(* CODESYS project Demo_MQTT.project

Project tree, tasks and I/O mapping:
  Device : P2CDS622, AutomationDirect.com, order no. n/a, version 1.1.8.0
    application Application
      libraries: Standard, 3.5.18.0 (System); StringUtils, 3.5.20.0 (System); VisuDialogs, * (System); MQTT Client SL, 1.9.0.0 (CODESYS); Web Socket Client SL, 1.9.0.0 (CODESYS); Net Base Services, 3.5.20.0 (CODESYS); BASIC, 3.31 (OSCAT)
      task MainTask (cyclic, interval t#20ms, priority 1) calls PRG
      task VISU_TASK (cyclic, interval 100 ms, priority 31) calls VisuElems.Visu_Prg
      program PRG [CFC]
      visualisation Visualization
      text list QoSTextlist
      function TerminateString [ST]
      image pool ImagePool
      text list ModeTextList
      text list VersionTextList
    Base : P2-04B, AutomationDirect.com, order no. abc, version 1.1.8.0
      Module : P2-08SIM, AutomationDirect.com, order no. P2-08SIM, version 0.0.2
          unmapped channels: Channels
      <Empty>
      <Empty>
      <Empty>
    P2CDS622_NetConfig : P2CDS622_NetConfig, AutomationDirect.com, order no. n/a, version 1.0.0.0
        settings: ET2: IP Address = [10,201,36,189]; ET2: Subnet Mask = [255,255,255,0]
  text list GlobalTextList
  5ce3da45-db07-42e7-a21c-a00fff4ed8f6|C:\Users\a.werner\Documents\background.jpg
*)

// Device/Application/PRG
// MQTT Client with visualization
PROGRAM PRG
VAR
	mqttClient : MQTT.MQTTClient; // Function block to establish a connection to a MQTT broker
	mqttPublisher : MQTT.MQTTPublish; // Function block to publish MQTT messages
	mqttPublisher2 : MQTT.MQTTPublish; // Function block to publish MQTT messages
	mqttSubscriber : MQTT.MQTTSubscribe; // Function block to subscribe MQTT topics
	mqttSubscriber2 : MQTT.MQTTSubscribe; // Function block to subscribe MQTT topics
	sHostname : STRING(255) := 'e737de6c210d405597c25f68240b4f2b.s2.eu.hivemq.cloud'; // My HiveMQ Hostname or ip address or URL (for WebSockets: ws:// or wss://)
	uiPort : UINT := 1883; // Port of the MQTT broker
	wsPublishTopic : WSTRING(1024) := ""; // Topic to publish a message
	wsPublishTopic2 : WSTRING(1024) := ""; // Topic to publish a message
	wsSubcribeTopicFilter : WSTRING(1024) := ""; // Topic filter to subcribe a topic
	wsSubcribeTopicFilter2 : WSTRING(1024) := ""; // Topic filter to subcribe a topic
	sWillMessage : STRING(1024); // The last will message
	sPublishMessage : STRING(1024) := ''; // The messsage to publish
	sPublishMessage2 : STRING(1024) := ''; // The messsage to publish
	sSubscribeMessage : STRING(4096); // Message buffer with the retrieved message  
	sSubscribeMessage2 : STRING(4096); // Message buffer with the retrieved message  
	rsPub1Error: RS; // Helper to publisher state
	rsPub1Done: RS; // Helper to publisher state
	rsPub2Error: RS; // Helper to publisher state
	rsPub2Done: RS; // Helper to publisher state
	eCommunicationMode : MQTT.COMMUNICATION_MODE := MQTT.COMMUNICATION_MODE.TCP; // Communication mode: TCP/IP or WebSockets
	eMQTTVersion : MQTT.MQTT_VERSION := MQTT.MQTT_VERSION.V3_1_1; // The MQTT protocol version

	// Example of connect properties (V5 only)
	mQTTConnectProperties : MQTT.MQTTConnectProperties := (
		udiSessionExpiryInterval := 10,
		udiMaximumPacketSize := MQTT.MQTTParam.g_udiMaxPacketSize,
		userProperties := 
			[
				(wsKey := "key1", wsValue := "value1"),
				(wsKey := "key2", wsValue := "value2"),	
				(wsKey := "key3", wsValue := "value3")
			]
	);
	
	// Example of will properties (V5 only)
	mQTTWillProperties : MQTT.MQTTWillProperties := (
		bPayloadFormatIndicator := 1, // 1: UTF-8, 0: Binary
		wsContentType := "text/plain",
		udiMessageExpiryInterval := 60,
		udiWillDelayInterval := 60,
		userProperties := 
		[
			(wsKey := "key1", wsValue := "value1"),
		 	(wsKey := "key2", wsValue := "value2"),	
			(wsKey := "key3", wsValue := "value3")
		]);
	
	// Example of publish properties (V5 only)
	mqTTPublishProperties : MQTT.MQTTPublishProperties := (
		bPayloadFormatIndicator := 1, // 1: UTF-8, 0: Binary
		wsContentType := "text/plain",
		udiMessageExpiryInterval := 60,
		userProperties := 
		[
			(wsKey := "key1", wsValue := "value1"),
		 	(wsKey := "key2", wsValue := "value2"),	
			(wsKey := "key3", wsValue := "value3")
		]
	);
	
	// Example of subscribe properties (V5 only)
	mQTTSubscribeProperties : MQTT.MQTTSubscribeProperties := (
		udiSubscriptionIdentifier := 4343,
		userProperties := 
		[
			(wsKey := "key1", wsValue := "value1"),
		 	(wsKey := "key2", wsValue := "value2"),	
			(wsKey := "key3", wsValue := "value3")
		],
		xNoLocalOption := FALSE
	);
	
	/// If you want to use client certificates, you can configure the connection via the TLS context.
	//
	// Example (static):
	//
	// _sCommonName : STRING := 'COMMON_NAME_OF_CERTIFICATE'; // CN of the certificate (common name). 
	// _sCipherList : NBS.CIPHER_LIST := STRUCT(psList := ADR('HIGH'), udiSize := 5); // Cipher string see https://www.openssl.org/docs/man1.1.1/man1/ciphers.html
	// _ciDefaultCertInfo : NBS.CERT_INFO := (psInfo := ADR(_sCommonName), udiSize := SIZEOF(_sCommonName)); // CN of the certificate (common name)
	
	// _tlsContext : NBS.TLSContext := (	sUseCaseName := _sCommonName, // A certificate is stored in the certificate store with the use case name. You can choose any name. Here we use the common name.
	//									ePurpose := NBS.PURPOSE.CLIENT_SIDE, // For client certificates set this to NBS.PURPOSE.CLIENT_SIDE
	//									sTLSVersion := '1.2', // The TLS version
	//									sCipherList := _sCipherList, // Set the cipher list
	//									sHostname := 'HOSTNAME_OF_THE_BROKER', // The hostname of the broker
	//									udiVerificationMode := 2, // 2 => Active Peer verification
	//									ciCertInfo := _ciDefaultCertInfo, // Set the cert info
	//									itfCertVerifer := 0); // 0 => No Verifier 
	// 
	// mqttClient : MQTT.MQTTClient := (itfTLSCOntext := _tlsContext);
    //
	// You can use the method TLSContext.SetInitialValue to set the context while runtime and set the context via the input itfTLSCOntext of the client FB.
END_VAR

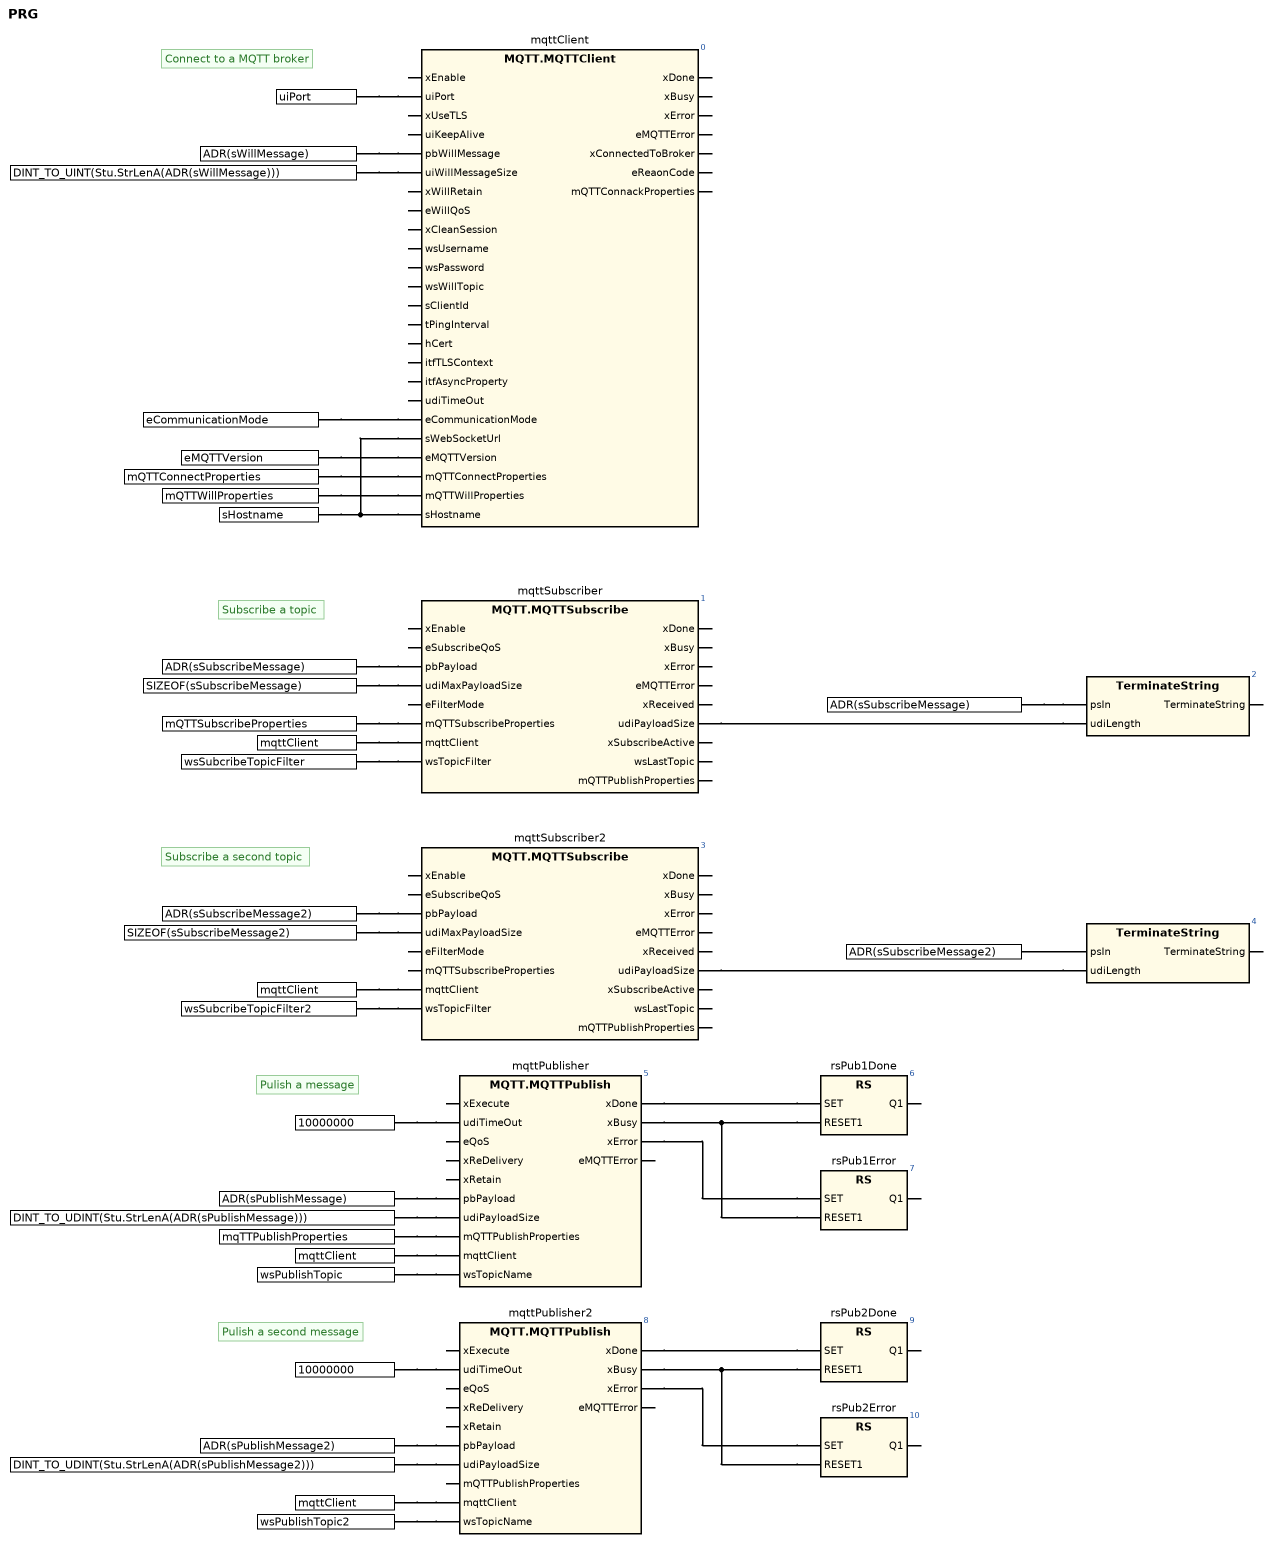
// Connect to a MQTT broker
mqttClient(
    uiPort := uiPort,
    pbWillMessage := ADR(sWillMessage),
    uiWillMessageSize := DINT_TO_UINT(Stu.StrLenA(ADR(sWillMessage))),
    eCommunicationMode := eCommunicationMode,
    sWebSocketUrl := sHostname,
    eMQTTVersion := eMQTTVersion,
    mQTTConnectProperties := mQTTConnectProperties,
    mQTTWillProperties := mQTTWillProperties,
    sHostname := sHostname); // MQTT.MQTTClient
// Subscribe a topic
mqttSubscriber(
    pbPayload := ADR(sSubscribeMessage),
    udiMaxPayloadSize := SIZEOF(sSubscribeMessage),
    mQTTSubscribeProperties := mQTTSubscribeProperties,
    mqttClient := mqttClient,
    wsTopicFilter := wsSubcribeTopicFilter); // MQTT.MQTTSubscribe
TerminateString(psIn := ADR(sSubscribeMessage), udiLength := mqttSubscriber.udiPayloadSize);
// Subscribe a second topic
mqttSubscriber2(
    pbPayload := ADR(sSubscribeMessage2),
    udiMaxPayloadSize := SIZEOF(sSubscribeMessage2),
    mqttClient := mqttClient,
    wsTopicFilter := wsSubcribeTopicFilter2); // MQTT.MQTTSubscribe
TerminateString(psIn := ADR(sSubscribeMessage2), udiLength := mqttSubscriber2.udiPayloadSize);
// Pulish a message
mqttPublisher(
    udiTimeOut := 10000000,
    pbPayload := ADR(sPublishMessage),
    udiPayloadSize := DINT_TO_UDINT(Stu.StrLenA(ADR(sPublishMessage))),
    mQTTPublishProperties := mqTTPublishProperties,
    mqttClient := mqttClient,
    wsTopicName := wsPublishTopic); // MQTT.MQTTPublish
rsPub1Done(SET := mqttPublisher.xDone, RESET1 := mqttPublisher.xBusy); // RS
rsPub1Error(SET := mqttPublisher.xError, RESET1 := mqttPublisher.xBusy); // RS
// Pulish a second message
mqttPublisher2(
    udiTimeOut := 10000000,
    pbPayload := ADR(sPublishMessage2),
    udiPayloadSize := DINT_TO_UDINT(Stu.StrLenA(ADR(sPublishMessage2))),
    mqttClient := mqttClient,
    wsTopicName := wsPublishTopic2); // MQTT.MQTTPublish
rsPub2Done(SET := mqttPublisher2.xDone, RESET1 := mqttPublisher2.xBusy); // RS
rsPub2Error(SET := mqttPublisher2.xError, RESET1 := mqttPublisher2.xBusy); // RS

END_PROGRAM

// Device/Application/TerminateString
// Terminates the STRING psIn at position udiLength
FUNCTION TerminateString : BOOL
VAR_INPUT
	psIn : POINTER TO BYTE; // Pointer to STRING
	udiLength : UDINT; // Length of psIn
END_VAR
VAR
END_VAR

psIn[udiLength] := 0;
TerminateString := TRUE;

END_FUNCTION

// Device/Application/Visualization
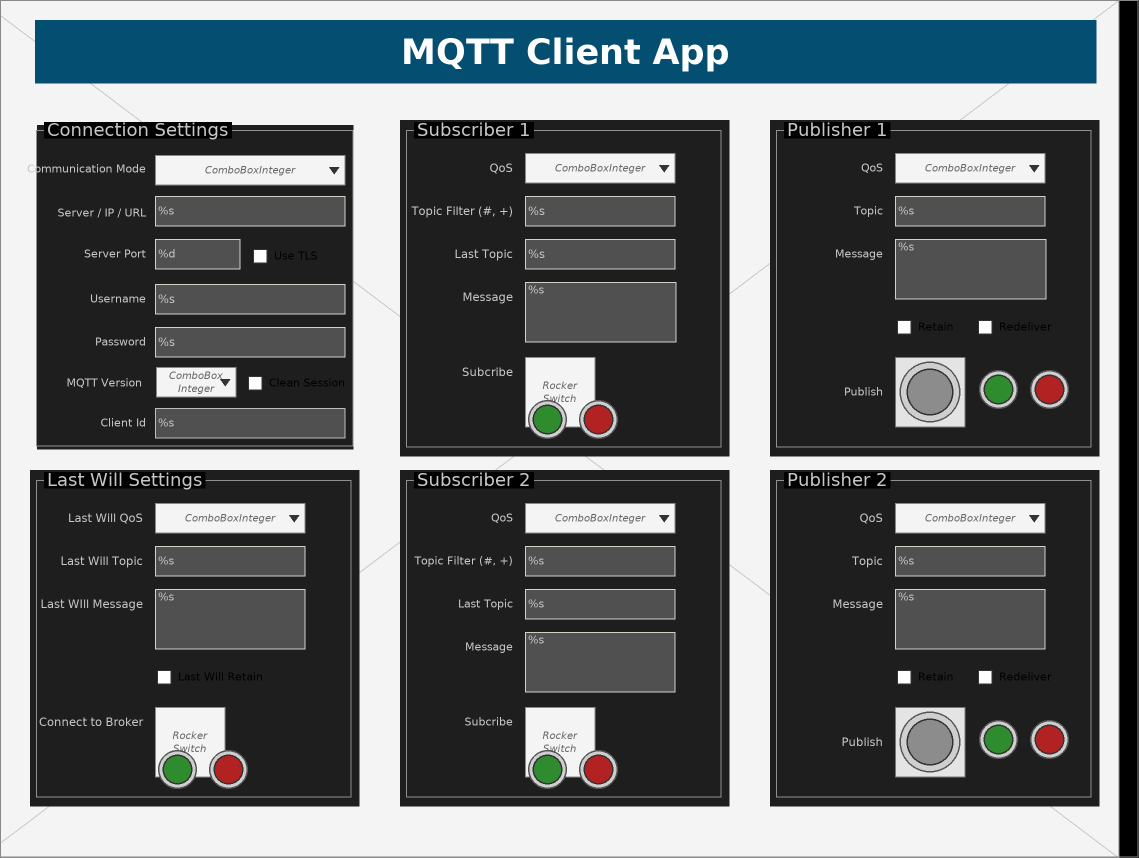
VISUALIZATION Visualization  // 1139x858
    Image (-20,0 1139x858), image: ImagePool.background
    Rectangle (37,125 316x324)
    Group (30,470 329x336)
        Rectangle (0,0 329x336)
        GroupBox (6,2 315x325), "Last Will Settings"
            ComboBoxInteger (119,31 150x30), variable: PRG.mqttClient.eWillQoS, text list: 'QoSTextlist'
        Label (16,33 100x30), "Last Will QoS"
        Textfield (125,76 150x30), "%s", text variable: PRG.mqttClient.wsWillTopic
            OnMouseClick: write the text variable via Default
        Label (16,76 100x30), "Last Will Topic"
        Textfield (125,119 150x60), "%s", text variable: PRG.sWillMessage
            OnMouseClick: write the text variable via Default
        Label (16,119 100x30), "Last WIll Message"
        Checkbox (125,192 150x30), "Last Will Retain", variable: PRG.mqttClient.xWillRetain
        Label (16,237 100x30), "Connect to Broker"
        RockerSwitch (125,237 70x70), variable: PRG.mqttClient.xEnable, behaviour: TOGGLE, style: Switch-RockerSwitch-Gray
        Lamp1 (125,277 45x45), variable: PRG.mqttClient.xConnectedToBroker, style: Lamp-Lamp1-Green
        Lamp1 (176,277 45x45), variable: PRG.mqttClient.xError, style: Lamp-Lamp1-Red
    Rectangle (770,120 329x336)
    GroupBox (776,122 315x325), "Publisher 1"
    ComboBoxInteger (895,153 150x30), variable: PRG.mqttPublisher.eQoS, text list: 'QoSTextlist'
    Label (786,153 100x30), "QoS"
    Textfield (895,196 150x30), "%s", text variable: PRG.wsPublishTopic
        OnMouseClick: write the text variable via Default
    Label (786,196 100x30), "Topic"
    Textfield (895,239 151x60), "%s", text variable: PRG.sPublishMessage
        OnMouseClick: write the text variable via Default
    Label (786,239 100x30), "Message"
    Checkbox (895,312 79x30), "Retain", variable: PRG.mqttPublisher.xRetain
    Checkbox (976,312 97x30), "Redeliver", variable: PRG.mqttPublisher.xReDelivery
    PushSwitch (895,357 70x70), variable: PRG.mqttPublisher.xExecute, input disabled if: NOT PRG.mqttClient.xConnectedToBroker, behaviour: TAP, style: Switch-PushSwitch-Gray
    Label (786,377 100x30), "Publish"
    Lamp1 (976,367 45x45), variable: PRG.rsPub1Done.Q1, style: Lamp-Lamp1-Green
    Lamp1 (1027,367 45x45), variable: PRG.rsPub1Error.Q1, style: Lamp-Lamp1-Red
    Group (770,470 329x336)
        Rectangle (0,0 329x336)
        GroupBox (6,2 315x325), "Publisher 2"
        ComboBoxInteger (125,33 150x30), variable: PRG.mqttPublisher2.eQoS, text list: 'QoSTextlist'
        Label (16,33 100x30), "QoS"
        Textfield (125,76 150x30), "%s", text variable: PRG.wsPublishTopic2
            OnMouseClick: write the text variable via Default
        Label (16,76 100x30), "Topic"
        Textfield (125,119 150x60), "%s", text variable: PRG.sPublishMessage2
            OnMouseClick: write the text variable via Default
        Label (16,119 100x30), "Message"
        Checkbox (125,192 80x30), "Retain", variable: PRG.mqttPublisher2.xRetain
        Checkbox (206,192 80x30), "Redeliver", variable: PRG.mqttPublisher2.xReDelivery
        PushSwitch (125,237 70x70), variable: PRG.mqttPublisher2.xExecute, input disabled if: NOT PRG.mqttClient.xConnectedToBroker, behaviour: TAP, style: Switch-PushSwitch-Gray
        Label (16,257 100x30), "Publish"
        Lamp1 (206,247 45x45), variable: PRG.rsPub2Done.Q1, style: Lamp-Lamp1-Green
        Lamp1 (257,247 45x45), variable: PRG.rsPub2Error.Q1, style: Lamp-Lamp1-Red
    Group (400,470 329x336)
        Rectangle (0,0 329x336)
        GroupBox (6,2 315x325), "Subscriber 2"
        ComboBoxInteger (125,33 150x30), variable: PRG.mqttSubscriber2.eSubscribeQoS, text list: 'QoSTextlist'
        Label (16,33 100x30), "QoS"
        Textfield (125,76 150x30), "%s", text variable: PRG.wsSubcribeTopicFilter2
            OnMouseClick: write the text variable via Default
        Label (16,76 100x30), "Topic Filter (#, +)"
        Textfield (125,162 150x60), "%s", text variable: PRG.sSubscribeMessage2
        Label (16,162 100x30), "Message"
        RockerSwitch (125,237 70x70), variable: PRG.mqttSubscriber2.xEnable, input disabled if: NOT PRG.mqttClient.xConnectedToBroker, behaviour: TOGGLE, style: Switch-RockerSwitch-Gray
        Label (16,237 100x30), "Subcribe"
        Lamp1 (125,277 45x45), variable: PRG.mqttSubscriber2.xSubscribeActive, style: Lamp-Lamp1-Green
        Lamp1 (176,277 45x45), variable: PRG.mqttSubscriber2.xError, style: Lamp-Lamp1-Red
        Label (16,119 100x30), "Last Topic"
        Textfield (125,119 150x30), "%s", text variable: PRG.mqttSubscriber2.wsLastTopic
    Group (400,120 329x336)
        Rectangle (0,0 329x336)
        GroupBox (6,2 315x325), "Subscriber 1"
        ComboBoxInteger (125,33 150x30), variable: PRG.mqttSubscriber.eSubscribeQoS, text list: 'QoSTextlist'
        Label (16,33 100x30), "QoS"
        Textfield (125,76 150x30), "%s", text variable: PRG.wsSubcribeTopicFilter
            OnMouseClick: write the text variable via Default
        Label (16,76 100x30), "Topic Filter (#, +)"
        Textfield (125,162 151x60), "%s", text variable: PRG.sSubscribeMessage
        Label (16,162 100x30), "Message"
        RockerSwitch (125,237 70x70), variable: PRG.mqttSubscriber.xEnable, input disabled if: NOT PRG.mqttClient.xConnectedToBroker, behaviour: TOGGLE, style: Switch-RockerSwitch-Gray
        Label (16,237 100x30), "Subcribe"
        Lamp1 (125,277 45x45), variable: PRG.mqttSubscriber.xSubscribeActive, style: Lamp-Lamp1-Green
        Lamp1 (176,277 45x45), variable: PRG.mqttSubscriber.xError, style: Lamp-Lamp1-Red
        Label (16,119 100x30), "Last Topic"
        Textfield (125,119 150x30), "%s", text variable: PRG.mqttSubscriber.wsLastTopic
    GroupBox (36,122 317x324), "Connection Settings"
        ComboBoxInteger (119,33 190x30), variable: PRG.eCommunicationMode, text list: 'ModeTextList'
        Label (-23,32 136x30), "Communication Mode"
        Textfield (119,74 190x30), "%s", text variable: PRG.sHostname
            OnMouseClick: write the text variable via Default
        Label (13,117 100x30), "Server Port", invisible if: PRG.eCommunicationMode = MQTT.COMMUNICATION_MODE.WEB_SOCKET
        Label (13,286 100x30), "Client Id"
        Textfield (119,286 190x30), "%s", text variable: PRG.mqttClient.sClientId
            OnMouseClick: write the text variable via Default
        Label (13,205 100x30), "Password"
        Textfield (119,205 190x30), "%s", text variable: PRG.mqttClient.wsPassword
            OnMouseClick: write the text variable via Default
        Label (13,162 100x30), "Username"
        Textfield (119,162 190x30), "%s", text variable: PRG.mqttClient.wsUsername
            OnMouseClick: write the text variable via Default
        Textfield (119,117 85x30), "%d", text variable: PRG.uiPort, invisible if: PRG.eCommunicationMode = MQTT.COMMUNICATION_MODE.WEB_SOCKET
            OnMouseClick: write the text variable via Default
        Label (-12,76 125x30), "Server / IP / URL"
        Checkbox (215,119 75x30), "Use TLS", variable: PRG.mqttClient.xUseTLS, invisible if: PRG.eCommunicationMode = MQTT.COMMUNICATION_MODE.WEB_SOCKET
        ComboBoxInteger (120,245 80x30), variable: PRG.eMQTTVersion, text list: 'VersionTextList'
        Label (23,246 86x30), "MQTT Version"
        Checkbox (210,246 103x30), "Clean Session", variable: PRG.mqttClient.xCleanSession
    Rectangle (35,20 1061x63), "MQTT Client App"
END_VISUALIZATION

(* text list QoSTextlist (id | default)
  0 | QoS 0
  1 | QoS 1
  2 | QoS 2
   |  *)

(* text list ModeTextList (id | default)
  0 | TCP/IP
  1 | WebSocket
   |  *)

(* text list VersionTextList (id | default)
  0 | 3.1.1
  1 | 5.0
   |  *)
